Fanuc TP program (LS listing): UP206.LS

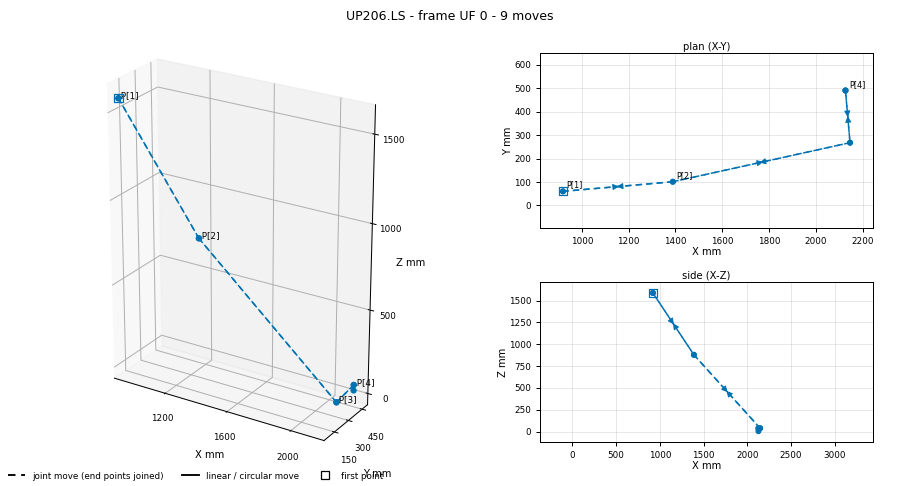
[picture p0: tool path of UP206.LS in frame UF 0, 9 of 9 moves have a stored position in this frame; points joined in program order, loops and branches not executed]
/PROG  UP206
/ATTR
OWNER		= SHIFT;
COMMENT		= "Prueba TCP SP1";
PROG_SIZE	= 3886;
CREATE		= DATE 16-10-11  TIME 00:31:40;
MODIFIED	= DATE 17-02-11  TIME 03:08:44;
FILE_NAME	= UP210;
VERSION		= 0;
LINE_COUNT	= 16;
MEMORY_SIZE	= 7494;
PROTECT		= READ_WRITE;
TCD:  STACK_SIZE	= 500,
      TASK_PRIORITY	= 50,
      TIME_SLICE	= 0,
      BUSY_LAMP_OFF	= 0,
      ABORT_REQUEST	= 0,
      PAUSE_REQUEST	= 0;
DEFAULT_GROUP	= 1,1,1,1,*;
CONTROL_CODE	= 00000000 00000000;
/APPL
/MN
   1:  UTOOL_NUM=24 ;
   2:  UFRAME_NUM=0 ;
   3:  PAYLOAD[1] ;
   4:J P[1] 100% CNT0 ACC100 TB    .10sec,P-SPS    ;
      1:  TC_ONLINE (ON) ;
      2:  DO[23]=OFF ;
      3:  CALL MAKRO050    ;
      4:  WAIT (DO[11])    ;
      5:  WAIT (DI[23])    ;
      6:  DO[23]=ON ;
      7:  TC_ONLINE (DO[11] AND M[2] AND M[30] AND M[31] AND M[33] AND M[35] AND M[37] AND M[39] AND M[41] AND M[95] AND M[96]) ;
       ------ ;
   5:J P[2] 100% CNT100 ACC100 TB   0.00sec,P-SPS    ;
      1:  TC_ONLINE (DO[11] AND M[2] AND M[30] AND M[31] AND M[33] AND M[35] AND M[37] AND M[39] AND M[41] AND M[95] AND M[96]) ;
       ------ ;
   6:J P[3] 100% CNT100 ACC100 TB   0.00sec,P-SPS    ;
      1:  TC_ONLINE (DO[11] AND M[2] AND M[30] AND M[31] AND M[33] AND M[35] AND M[37] AND M[39] AND M[41] AND M[95] AND M[96]) ;
       ------ ;
   7:J P[4] 100% CNT0 ACC100 TB    .10sec,P-SPS    ;
      1:  TC_ONLINE (ON) ;
      2:  DO[23]=OFF ;
      3:  WAIT (DI[23])    ;
      4:  DO[23]=ON ;
      5:  TC_ONLINE (DO[11] AND M[2] AND M[30] AND M[31] AND M[33] AND M[35] AND M[37] AND M[39] AND M[41] AND M[95] AND M[96]) ;
       ------ ;
   8:  !Posicion Prueba TCP ;
   9:  !SP1 ;
  10:  !X=2126.017 Y=490.973 Z=5.968 ;
  11:  !W=-179.917 P=3.073 R=-86.565 ;
  12:L P[5] 400mm/sec CNT0 ACC100 TB    .10sec,P-SPS    ;
      1:  TC_ONLINE (ON) ;
      2:  DO[23]=OFF ;
      3:  WAIT (DI[17])    ;
      4:  WAIT (DI[23])    ;
      5:  DO[23]=ON ;
      6:  TC_ONLINE (DO[11] AND M[2] AND M[30] AND M[31] AND M[33] AND M[35] AND M[37] AND M[39] AND M[41] AND M[95] AND M[96]) ;
       ------ ;
  13:L P[6] 400mm/sec CNT0 ACC100 TB    .10sec,P-SPS    ;
      1:  TC_ONLINE (ON) ;
      2:  DO[23]=OFF ;
      3:  WAIT (DI[23])    ;
      4:  DO[23]=ON ;
      5:  TC_ONLINE (DO[11] AND M[2] AND M[30] AND M[31] AND M[33] AND M[35] AND M[37] AND M[39] AND M[41] AND M[95] AND M[96]) ;
       ------ ;
  14:J P[7] 100% CNT100 ACC100 TB   0.00sec,P-SPS    ;
      1:  TC_ONLINE (DO[11] AND M[2] AND M[30] AND M[31] AND M[33] AND M[35] AND M[37] AND M[39] AND M[41] AND M[95] AND M[96]) ;
       ------ ;
  15:J P[8] 100% CNT100 ACC100 TB   0.00sec,P-SPS    ;
      1:  TC_ONLINE (DO[11] AND M[2] AND M[30] AND M[31] AND M[33] AND M[35] AND M[37] AND M[39] AND M[41] AND M[95] AND M[96]) ;
       ------ ;
  16:J P[9] 100% CNT0 ACC100 TB    .10sec,P-SPS    ;
      1:  TC_ONLINE (ON) ;
      2:  DO[23]=OFF ;
      3:  WAIT (DI[23])    ;
      4:  DO[23]=ON ;
      5:  TC_ONLINE (DO[11] AND M[2] AND M[30] AND M[31] AND M[33] AND M[35] AND M[37] AND M[39] AND M[41] AND M[95] AND M[96]) ;
       ------ ;
/POS
P[1]{
   GP1:
	UF : 0, UT : 24,		CONFIG : 'N U T, 0, 0, 1',
	X =   919.379  mm,	Y =    60.188  mm,	Z =  1586.575  mm,
	W =  -170.243 deg,	P =    39.286 deg,	R =  -167.434 deg
   GP2:
	UF : 4, UT : 24,
	J1=   100.000  mm
   GP3:
	UF : 0, UT : 24,
	J1=     0.000  mm
   GP4:
	UF : 0, UT : 24,
	J1=     0.000  mm
};
P[2]{
   GP1:
	UF : 0, UT : 24,		CONFIG : 'N U T, 0, 0, 1',
	X =  1388.517  mm,	Y =   101.381  mm,	Z =   879.364  mm,
	W =  -173.064 deg,	P =    -1.222 deg,	R =  -119.075 deg
   GP2:
	UF : 0, UT : 24,
	J1=   100.000  mm
   GP3:
	UF : 0, UT : 24,
	J1=     0.000  mm
   GP4:
	UF : 0, UT : 24,
	J1=     0.000  mm
};
P[3]{
   GP1:
	UF : 0, UT : 24,		CONFIG : 'N U T, 0, 0, 1',
	X =  2145.512  mm,	Y =   268.144  mm,	Z =    39.616  mm,
	W =  -179.917 deg,	P =     3.073 deg,	R =   -86.564 deg
   GP2:
	UF : 0, UT : 24,
	J1=   100.000  mm
   GP3:
	UF : 0, UT : 24,
	J1=     0.000  mm
   GP4:
	UF : 0, UT : 24,
	J1=     0.000  mm
};
P[4]{
   GP1:
	UF : 0, UT : 24,		CONFIG : 'N U T, 0, 0, 1',
	X =  2126.017  mm,	Y =   490.973  mm,	Z =    39.616  mm,
	W =  -179.917 deg,	P =     3.073 deg,	R =   -86.565 deg
   GP2:
	UF : 0, UT : 24,
	J1=   100.000  mm
   GP3:
	UF : 0, UT : 24,
	J1=     0.000  mm
   GP4:
	UF : 0, UT : 24,
	J1=     0.000  mm
};
P[5]{
   GP1:
	UF : 0, UT : 24,		CONFIG : 'N U T, 0, 0, 1',
	X =  2126.017  mm,	Y =   490.973  mm,	Z =     5.968  mm,
	W =  -179.917 deg,	P =     3.073 deg,	R =   -86.565 deg
   GP2:
	UF : 0, UT : 24,
	J1=   100.000  mm
   GP3:
	UF : 0, UT : 24,
	J1=     0.000  mm
   GP4:
	UF : 0, UT : 24,
	J1=     0.000  mm
};
P[6]{
   GP1:
	UF : 0, UT : 24,		CONFIG : 'N U T, 0, 0, 1',
	X =  2126.017  mm,	Y =   490.973  mm,	Z =    39.616  mm,
	W =  -179.917 deg,	P =     3.073 deg,	R =   -86.565 deg
   GP2:
	UF : 0, UT : 24,
	J1=   100.000  mm
   GP3:
	UF : 0, UT : 24,
	J1=     0.000  mm
   GP4:
	UF : 0, UT : 24,
	J1=     0.000  mm
};
P[7]{
   GP1:
	UF : 0, UT : 24,		CONFIG : 'N U T, 0, 0, 1',
	X =  2145.512  mm,	Y =   268.144  mm,	Z =    39.616  mm,
	W =  -179.917 deg,	P =     3.073 deg,	R =   -86.564 deg
   GP2:
	UF : 0, UT : 24,
	J1=   100.000  mm
   GP3:
	UF : 0, UT : 24,
	J1=     0.000  mm
   GP4:
	UF : 0, UT : 24,
	J1=     0.000  mm
};
P[8]{
   GP1:
	UF : 0, UT : 24,		CONFIG : 'N U T, 0, 0, 1',
	X =  1388.517  mm,	Y =   101.381  mm,	Z =   879.364  mm,
	W =  -173.064 deg,	P =    -1.222 deg,	R =  -119.075 deg
   GP2:
	UF : 0, UT : 24,
	J1=   100.000  mm
   GP3:
	UF : 0, UT : 24,
	J1=     0.000  mm
   GP4:
	UF : 0, UT : 24,
	J1=     0.000  mm
};
P[9]{
   GP1:
	UF : 0, UT : 24,		CONFIG : 'N U T, 0, 0, 1',
	X =   919.379  mm,	Y =    60.188  mm,	Z =  1586.575  mm,
	W =  -170.243 deg,	P =    39.286 deg,	R =  -167.434 deg
   GP2:
	UF : 4, UT : 24,
	J1=   100.000  mm
   GP3:
	UF : 0, UT : 24,
	J1=     0.000  mm
   GP4:
	UF : 0, UT : 24,
	J1=     0.000  mm
};
/END
